(* TLS/PSK configuration *)
{attribute 'no_explicit_call':='Direct call not allowed for type FB_TlsConfig'}
{attribute 'no_assign'}
FUNCTION_BLOCK FB_TlsConfig
VAR
	_pskKey       : ARRAY[0..TCPADS_TLS_MAX_PSK_KEY_SIZE] OF BYTE;
	_pskKeyLen    : UDINT:=0;
	_sIdentity    : STRING(TCPADS_TLS_PSK_IDENTITY_SIZE);
	_sCaPath      : STRING(TCPADS_TLS_CERTIFICATE_PATH_SIZE);
	_sCrlPath     : STRING(TCPADS_TLS_CERTIFICATE_PATH_SIZE);
	_sCertPath    : STRING(TCPADS_TLS_CERTIFICATE_PATH_SIZE);
	_sKeyPath     : STRING(TCPADS_TLS_CERTIFICATE_PATH_SIZE);
	_sKeyPwd      : STRING(TCPADS_TLS_KEY_PASSWORD_SIZE);
	_listenFlags  : ST_TlsListenFlags:=DEFAULT_TLSLISTENFLAGS;
	_connectFlags : ST_TlsConnectFlags:=DEFAULT_TLSCONNECTFLAGS;
END_VAR

(* Adds CA certificate path *)
METHOD FINAL AddCa
VAR_INPUT
	sCaPath : STRING(TCPADS_TLS_CERTIFICATE_PATH_SIZE);
END_VAR
_sCaPath:=sCaPath;
END_METHOD

(* Adds certificate path *)
METHOD FINAL AddCert
VAR_INPUT
	sCertPath: STRING(TCPADS_TLS_CERTIFICATE_PATH_SIZE);
	sKeyPath: STRING(TCPADS_TLS_CERTIFICATE_PATH_SIZE);
	sKeyPwd: STRING(TCPADS_TLS_KEY_PASSWORD_SIZE);
END_VAR
_sCertPath:=sCertPath;
_sKeyPath:=sKeyPath;
_sKeyPwd:=sKeyPwd;
END_METHOD

METHOD FINAL AddConnectFlags
VAR_INPUT
	flags : ST_TlsConnectFlags;
END_VAR
_connectFlags:=flags;
END_METHOD

(* Adds certificate revocation list path *)
METHOD FINAL AddCrl
VAR_INPUT
	sCrlPath : STRING(TCPADS_TLS_CERTIFICATE_PATH_SIZE);
END_VAR
_sCrlPath:=sCrlPath;
END_METHOD

METHOD FINAL AddListenFlags
VAR_INPUT
	flags : ST_TlsListenFlags;
END_VAR
_listenFlags:=flags;
END_METHOD

(* Adds PSK and PSK identity *)
METHOD FINAL AddPsk
VAR_IN_OUT
	key : ARRAY[*] OF BYTE;
END_VAR
VAR_INPUT
	sIdentity : STRING(TCPADS_TLS_PSK_IDENTITY_SIZE);
END_VAR
_pskKeyLen:=MIN(DINT_TO_UDINT(UPPER_BOUND(key, 1) - LOWER_BOUND(key, 1) + 1), TCPADS_TLS_MAX_PSK_KEY_SIZE, SIZEOF(_pskKey));
MEMCPY(ADR(_pskKey[0]), ADR(key[LOWER_BOUND(key, 1)]), _pskKeyLen);
_sIdentity:=sIdentity;
END_METHOD

METHOD FINAL Clear
_sIdentity:='';
_pskKeyLen:=0;
MEMSET(ADR(_pskKey[0]), 0, SIZEOF(_pskKey));
_sCaPath:='';
_sCertPath:='';
_sKeyPath:='';
_sKeyPwd:='';
_sCrlPath:='';
_listenFlags:=DEFAULT_TLSLISTENFLAGS;
_connectFlags:=DEFAULT_TLSCONNECTFLAGS;
END_METHOD

PROPERTY FINAL connectFlags : ST_TlsConnectFlags
GET
connectFlags:=_connectFlags;
END_GET
END_PROPERTY

PROPERTY FINAL listenFlags : ST_TlsListenFlags
GET
listenFlags:=_listenFlags;
END_GET
END_PROPERTY

(* Pointer to first PSK key byte *)
PROPERTY FINAL pskKey : PVOID
GET
pskKey:=SEL(_pskKeyLen = 0, ADR(_pskKey[0]), 0);
END_GET
END_PROPERTY

(* Byte size of PSK key *)
PROPERTY FINAL pskKeyLen : UDINT(0..TCPADS_TLS_MAX_PSK_KEY_SIZE)
GET
pskKeyLen:=_pskKeyLen;
END_GET
END_PROPERTY

(* CA certificate path *)
PROPERTY FINAL sCaPath : STRING(TCPADS_TLS_CERTIFICATE_PATH_SIZE)
GET
sCaPath:=_sCaPath;
END_GET
END_PROPERTY

(* Certificate path *)
PROPERTY FINAL sCertPath : STRING(TCPADS_TLS_CERTIFICATE_PATH_SIZE)
GET
sCertPath:=_sCertPath;
END_GET
END_PROPERTY

(* Certificate revocation list path *)
PROPERTY FINAL sCrlPath : STRING(TCPADS_TLS_CERTIFICATE_PATH_SIZE)
GET
sCrlPath:=_sCrlPath;
END_GET
END_PROPERTY

(* PSK key identity *)
PROPERTY FINAL sIdentity : STRING(TCPADS_TLS_PSK_IDENTITY_SIZE)
GET
sIdentity:=_sIdentity;
END_GET
END_PROPERTY

(* Certificate key path *)
PROPERTY FINAL sKeyPath : STRING(TCPADS_TLS_CERTIFICATE_PATH_SIZE)
GET
sKeyPath:=_sKeyPath;
END_GET
END_PROPERTY

(* Certificate key password *)
PROPERTY FINAL sKeyPwd : STRING(TCPADS_TLS_KEY_PASSWORD_SIZE)
GET
sKeyPwd:=_sKeyPwd;
END_GET
END_PROPERTY

END_FUNCTION_BLOCK

(* stored: Version 1.1.0.1
   POU FB_TlsConfig: Id {93e96eff-fdb4-46dc-acd8-f9caf2220236}, SpecialFunc None
   Method AddCa: Id {1961e798-3f87-47ac-96f6-547d20f17058}
   Method AddCert: Id {a02414a8-af73-46aa-b7f1-9ddd84dd131d}
   Method AddConnectFlags: Id {0ecfc7d8-b506-42b2-b1a2-18fbf7003f77}
   Method AddCrl: Id {53ba7074-e1c8-411c-8d89-9cb56fdeedc1}
   Method AddListenFlags: Id {e5a3d6e3-5e7e-4bb0-9ba5-8145ae2ea7b0}
   Method AddPsk: Id {fe01aa1a-6244-4223-a587-9e1014330cc9}
   Method Clear: Id {b03107d9-5004-4d9e-a30c-c180f2a31e61}
   Property connectFlags: Id {8c8dd301-8861-4876-8fd2-4f2e756d91d5}
   Get Get: Id {a1b970a4-7622-416e-8940-f3aab3e82f4c}
   Property listenFlags: Id {a625f6c6-3762-4ade-a6a8-4457726e56ed}
   Get Get: Id {ad9cd4a1-95ef-442b-b395-d79ba11aa2ee}
   Property pskKey: Id {e3ea9e26-aa80-47bc-8a69-329a2a57f84c}
   Get Get: Id {d81c707f-5605-499f-bd67-943e24e1cd18}
   Property pskKeyLen: Id {3c3b4625-a194-4b92-8df5-1fe2ff9d9882}
   Get Get: Id {002ec0d2-217b-4c08-ba6e-13497e3cb68c}
   Property sCaPath: Id {d0808b44-c122-4a24-b79a-e479e00e92ed}
   Get Get: Id {5b540fb9-1611-483e-9e05-4cb935597a25}
   Property sCertPath: Id {a34d6a2e-8ecd-4758-8991-07fd960798ea}
   Get Get: Id {b1b28fe8-aadf-4756-979e-be4cff5db0f1}
   Property sCrlPath: Id {93714f42-87b4-4cf0-8647-a68ad64c7083}
   Get Get: Id {96f75915-94d0-461f-9ca1-963bf86812e4}
   Property sIdentity: Id {6de5b960-ba34-4e5d-bbd3-b9df137e3c8e}
   Get Get: Id {446878f3-d332-4b9b-aa63-05ba5664c0b9}
   Property sKeyPath: Id {31e05108-ffd0-47bf-8fc1-dac58ea05be4}
   Get Get: Id {d3b3daa3-f1c8-44c4-af02-2d5229ec4be6}
   Property sKeyPwd: Id {fb7ad24f-2a13-4ab3-93ef-c770f12fc9fb}
   Get Get: Id {cc53f680-3374-480e-b94b-3271d20a6a81} *)
